{attribute 'qualified_only'}
{attribute 'strict'}
TYPE EComparisonType :
(
	none := 0,
	equals := 1,
	not_equal := 2,
	greater := 3,
	less := 4,
	greater_eq := 5,
	less_eq := 6
);
END_TYPE

(* stored: Version 1.1.0.1, ProductVersion 3.1.4024.9
   DUT EComparisonType: Id {e0779ba4-ab3e-4ee9-9c01-a83fd9e8558c} *)
